FUNCTION_BLOCK EL1012
VAR
	_io : EL1xx2_Data;
	{attribute addProperty Name "WcState"}
	_wcState : WcStateInputToggle;
	{attribute addProperty Name "Info data"}
	_infoData : InfoDataBase;
END_VAR

PROPERTY IO : REFERENCE TO EL1xx2_Data
GET
IO REF= _io;
END_GET
END_PROPERTY

PROPERTY WcState : REFERENCE TO WcStateInputToggle
GET
WcState REF= _wcState;
END_GET
END_PROPERTY

END_FUNCTION_BLOCK

(* stored: Version 1.1.0.1, ProductVersion 3.1.4024.9
   POU EL1012: Id {b5b6fd38-184d-02bc-0b68-66c70f1acd32}, SpecialFunc None
   Property IO: Id {34dabf44-78de-0737-0e49-501ae5a77921}
   Get Get: Id {6bb4c8d1-ded3-0cf0-344c-7bcfa3110a03}
   Property WcState: Id {ce787ce7-a0fc-06c0-125d-0241105ba50f}
   Get Get: Id {b7b083a8-f1cd-04a0-2b7c-7e7ddde1aff6} *)
